TYPE DUT_HMI_03_MANUALS :
STRUCT
	PS : ARRAY[0..CNC.NUM_MAX_MANUALS_03-1] OF BOOL;
	LS : ARRAY[0..CNC.NUM_MAX_MANUALS_03-1] OF BOOL;
END_STRUCT
END_TYPE

(* stored: Version 1.1.0.1, ProductVersion 3.1.4024.13
   DUT DUT_HMI_03_MANUALS: Id {ef4787c5-4e09-4931-843d-7079b397b690} *)
